// TwinCAT 3 PLC project ExecuteProgram
// ProgramVersion: 3.1.4022.3
// libraries:
//   BeckhoffHttpClient, * (fbarresi)
//   Tc2_Standard, * (Beckhoff Automation GmbH)
//   Tc2_System, * (Beckhoff Automation GmbH)
//   Tc2_Utilities, * (Beckhoff Automation GmbH)
//   Tc3_Module, * (Beckhoff Automation GmbH)
// project tree:
//   DUTs/ Json.TcDUT, unterJson.TcDUT
//   GVLs/ GVL.TcGVL
//   POUs/ MAIN.TcPOU
//   / programm.TcTTO
// real-time tasks:
//   TASK programm: cycle T#1ms, priority 20, ADS port 350

CONFIGURATION ExecuteProgram
    RESOURCE PLC ON TwinCAT3
        TASK programm(INTERVAL := T#1ms, PRIORITY := 20);
        PROGRAM MAIN WITH programm : MAIN;
    END_RESOURCE
END_CONFIGURATION

// ---- DUTs/Json.TcDUT
TYPE Json :
STRUCT
	{attribute 'json' := 'message'}
	Messaggio : STRING;
	response : INT;
	{attribute 'json' := 'status'}
	stato : STRING;
	{attribute 'json' := 'Numbers'}
	numeri : ARRAY[1..10] OF DINT := [1,2,3,4,5,6,7,8,9,10];
	{attribute 'json'}
	child : unterJson;
	{attribute 'json'}
	children : ARRAY [0..3] OF unterJson;
END_STRUCT
END_TYPE

// ---- DUTs/unterJson.TcDUT
TYPE unterJson :
STRUCT
	{attribute 'json' := 'message'}
	Messaggio : STRING;
	response : INT;
	{attribute 'json' := 'status'}
	stato : STRING;
	{attribute 'json' := 'doubles'}
	ArrayDouble : ARRAY[1..10] OF LREAL := [1.1,2.1,3.1,4.1,5.1,6.1,7.1,8.1,9.1,10.1];
END_STRUCT
END_TYPE

// ---- GVLs/GVL.TcGVL
{attribute 'qualified_only'}
VAR_GLOBAL
	{attribute 'federico' := 'The best'}
	Body : ARRAY [1..10] OF STRING;
	test : json;
END_VAR

// ---- POUs/MAIN.TcPOU
PROGRAM MAIN
VAR
	client : HttpClient;
END_VAR

client();

END_PROGRAM
